(* CoDeSys 2.3 export: V3_ABS.EXP *)

(* POU Mathematical/Vektormathematik/V3_ABS, ST *)
FUNCTION V3_ABS : REAL
VAR_INPUT
	A : Vector_3;
END_VAR


(*
version 1.0	11 dec 2007
programmer 	hugo
tested by		tobias

this function calculates the length of a vectors in a 3 dimensional space

*)
V3_ABS := SQRT(A.X * A.X + A.Y * A.Y + A.Z * A.Z);


(* revision history
hm		11 dec 2007	rev 1.0
	original version

*)
END_FUNCTION
